(* PLC project BE_Framework BA.project, CODESYS CODESYS V3.5 SP13 Patch 2 *)
(* stored: creationDateTime 2018-11-30T22:01:10.149683, modificationDateTime 2018-11-30T22:00:52.5249251 *)

PROGRAM LB01_FF1_Analog_ST
VAR
	local:strFan_Analog;
	localGP:strSensor2_Regulator;
	ControlFan: _BE_Fan;
	FbRegulator: _BE_Regulator;
	_BE_Fan2: _BE_Fan_2;
	reset_en: RS;
	AlarmFbAl03: _BE_AlarmAckRequired;
	AlarmFbAl02: _BE_AlarmAckRequired;
	fb_OperationalTime: _BE_OperationalTime;
	ackAl01: BOOL;
	ackAl02: BOOL;
	fanGuardOk: BOOL;
END_VAR

            //Struct ->> local
LB01.FF1 := local;
LB01.GP22 := localGP;
LB01.GP23.V := fanGuardOk;

//Fan

//Alarm

//Regulator

//Operational time
fb_OperationalTime(Operating := local.CMD, MinutePulse := SYS_MinutePulse, ResetOperatingTime := local.RST, ResetStarts := local.RST);
local.PV2 := fb_OperationalTime.TotalMinutes;
local.PV1 := fb_OperationalTime.TotalHours;
local.PV3 := fb_OperationalTime.StartsTotal;

//Local --> STRUCT
local := LB01.FF1;
localGP := LB01.GP21;


          
END_PROGRAM
